Fanuc KAREL source: kb00155.KL

-- PROVISIONAL review KL for V1013-1; original PC SHA256 2c3e98de5861c9ad412af2e34c44611333ca52b608da52c33f8c9602a9b13bb0
-- Incomplete behavior may be omitted. Consult companion uncertainty JSON. Do not deploy.
PROGRAM KB00155
%NOLOCKGROUP
BEGIN
  -- UNRESOLVED_PC offsets 5-14; opcodes 3F,75
  -- UNRESOLVED_PC offsets 19-26; opcodes 9D,23
  -- UNRESOLVED_PC offsets 31-49; opcodes 27,22,2A,22,31
  -- UNRESOLVED_PC offsets 54-58; opcodes 7F
END KB00155
